TYPE InfluxData :
STRUCT
	CycleCount : UDINT;
	CycleTime : UDINT;
	LastExecTime: UDINT;
END_STRUCT
END_TYPE

(* stored: Version 1.1.0.1, ProductVersion 3.1.4024.3
   DUT InfluxData: Id {364eb6fb-b337-44ff-8300-53525e7c3755} *)
